// P1 - E_Errors2_ReactorSet
// Rev 1.0 - October 31, 2024

TYPE E_Errors2_ReactorSet :
(
	errTBD								:= 0
);
END_TYPE

(* stored: Version 1.1.0.1, ProductVersion 3.1.4024.13
   DUT E_Errors2_ReactorSet: Id {e7f4f99f-0e17-49c1-bbaa-51e4b5c885ca} *)
